SUBAPPLICATION SubApp (* Subapplication Type *)
  (* Standard: 61499-2 *)
  (* Version 1.0, 2022-12-28, kirill *)
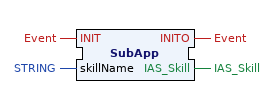
  EVENT_INPUT
    INIT;
  END_EVENT
  EVENT_OUTPUT
    INITO;
  END_EVENT
  VAR_INPUT
    skillName : STRING;
  END_VAR
  PLUGS
    IAS_Skill : IAS_Skill;
  END_PLUGS
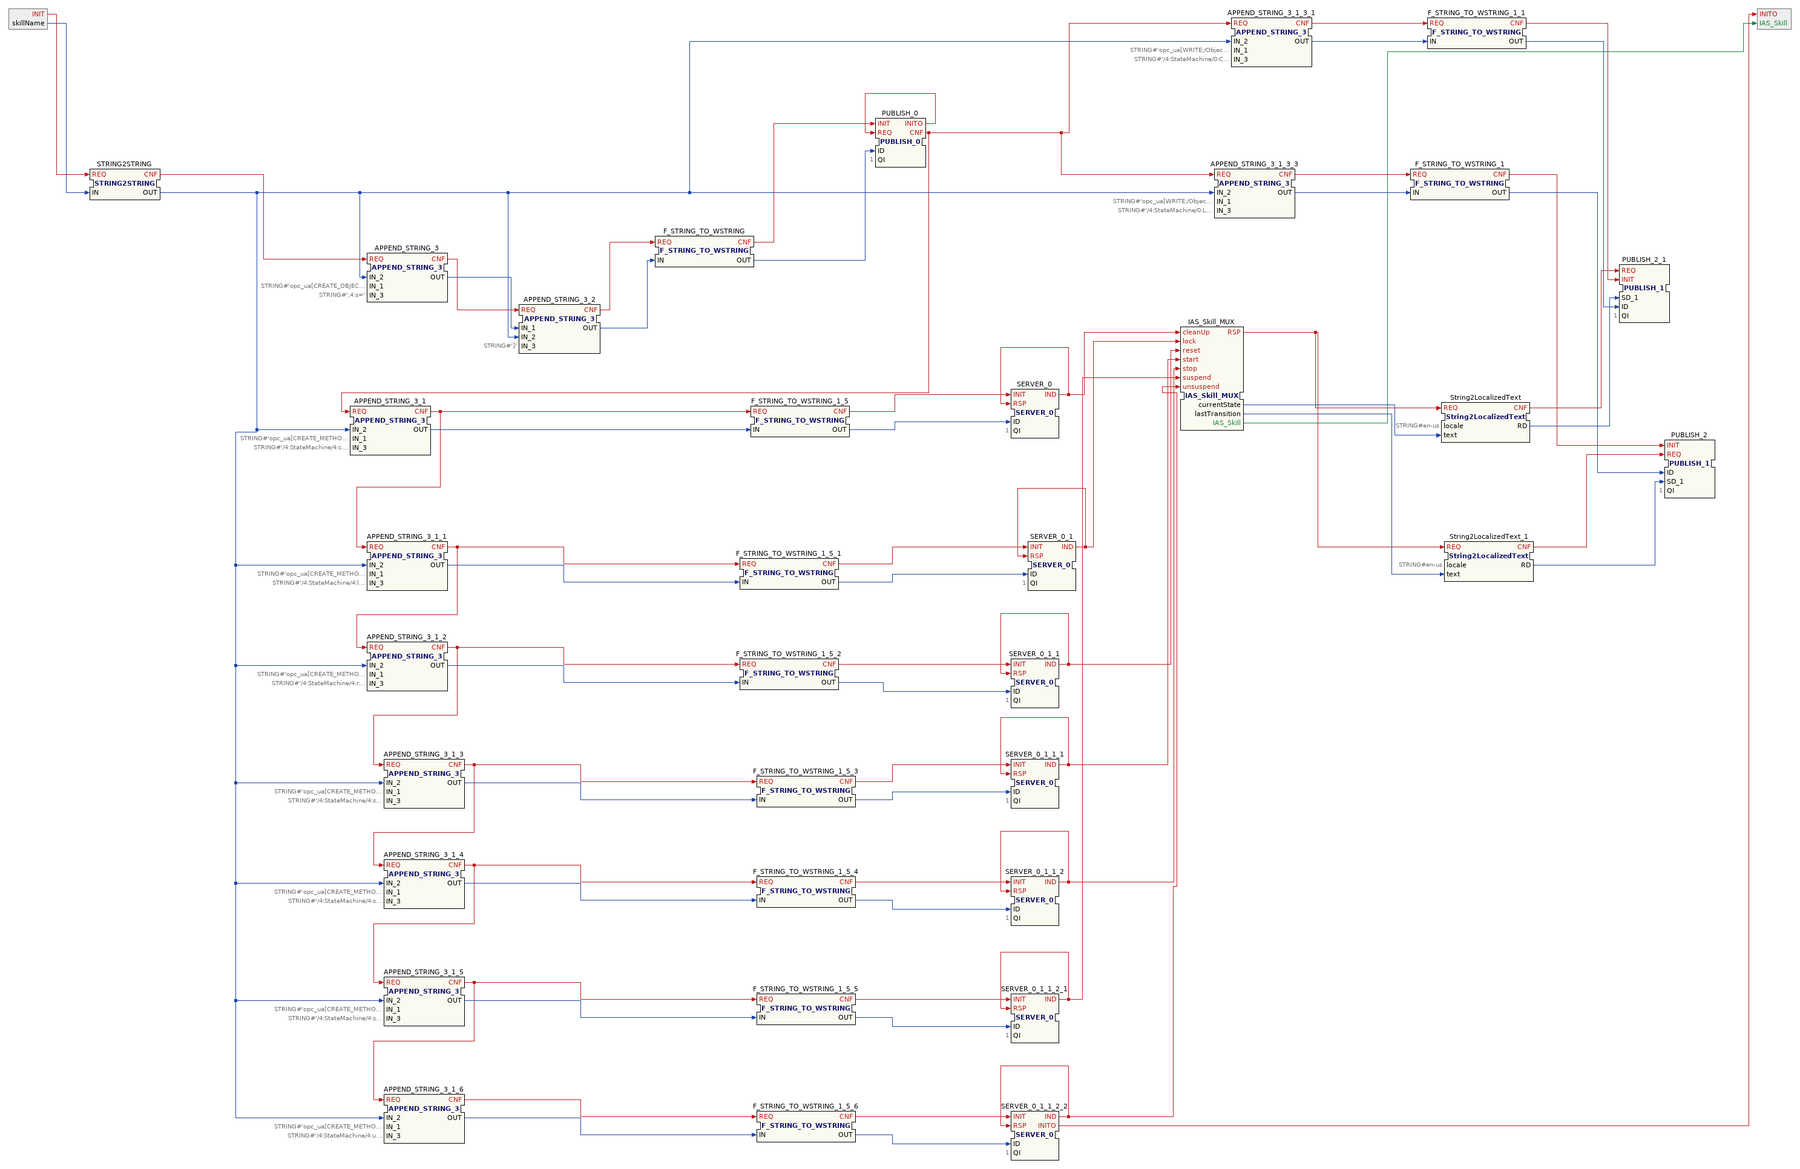
  FBS
    SERVER_0 : SERVER_0(QI := 1);
    APPEND_STRING_3 : APPEND_STRING_3(IN_1 := STRING#'opc_ua[CREATE_OBJECT;,i=58;/Objects/4:', IN_3 := STRING#',4:s=');
    PUBLISH_0 : PUBLISH_0(QI := 1);
    String2LocalizedText : String2LocalizedText(locale := STRING#en-us);
    STRING2STRING : STRING2STRING;
    SERVER_0_1_1_2 : SERVER_0(QI := 1);
    APPEND_STRING_3_1_3_1 : APPEND_STRING_3(IN_1 := STRING#'opc_ua[WRITE;/Objects/4:', IN_3 := STRING#'/4:StateMachine/0:CurrentState]');
    F_STRING_TO_WSTRING_1_5_1 : F_STRING_TO_WSTRING;
    APPEND_STRING_3_1_3_3 : APPEND_STRING_3(IN_1 := STRING#'opc_ua[WRITE;/Objects/4:', IN_3 := STRING#'/4:StateMachine/0:LastTransition]');
    F_STRING_TO_WSTRING_1_5 : F_STRING_TO_WSTRING;
    F_STRING_TO_WSTRING_1_1 : F_STRING_TO_WSTRING;
    IAS_Skill_MUX : IAS_Skill_MUX;
    APPEND_STRING_3_1_2 : APPEND_STRING_3(IN_1 := STRING#'opc_ua[CREATE_METHOD;/Objects/4:', IN_3 := STRING#'/4:StateMachine/4:reset]');
    SERVER_0_1_1_2_1 : SERVER_0(QI := 1);
    PUBLISH_2 : PUBLISH_1(QI := 1);
    SERVER_0_1_1_1 : SERVER_0(QI := 1);
    SERVER_0_1 : SERVER_0(QI := 1);
    APPEND_STRING_3_2 : APPEND_STRING_3(IN_3 := STRING#']');
    F_STRING_TO_WSTRING_1_5_5 : F_STRING_TO_WSTRING;
    SERVER_0_1_1 : SERVER_0(QI := 1);
    F_STRING_TO_WSTRING_1_5_3 : F_STRING_TO_WSTRING;
    APPEND_STRING_3_1_4 : APPEND_STRING_3(IN_1 := STRING#'opc_ua[CREATE_METHOD;/Objects/4:', IN_3 := STRING#'/4:StateMachine/4:stop]');
    APPEND_STRING_3_1_3 : APPEND_STRING_3(IN_1 := STRING#'opc_ua[CREATE_METHOD;/Objects/4:', IN_3 := STRING#'/4:StateMachine/4:start]');
    PUBLISH_2_1 : PUBLISH_1(QI := 1);
    APPEND_STRING_3_1_1 : APPEND_STRING_3(IN_1 := STRING#'opc_ua[CREATE_METHOD;/Objects/4:', IN_3 := STRING#'/4:StateMachine/4:lock]');
    F_STRING_TO_WSTRING_1_5_2 : F_STRING_TO_WSTRING;
    APPEND_STRING_3_1_6 : APPEND_STRING_3(IN_1 := STRING#'opc_ua[CREATE_METHOD;/Objects/4:', IN_3 := STRING#'/4:StateMachine/4:unsuspend]');
    F_STRING_TO_WSTRING : F_STRING_TO_WSTRING;
    SERVER_0_1_1_2_2 : SERVER_0(QI := 1);
    APPEND_STRING_3_1 : APPEND_STRING_3(IN_1 := STRING#'opc_ua[CREATE_METHOD;/Objects/4:', IN_3 := STRING#'/4:StateMachine/4:cleanUp]');
    F_STRING_TO_WSTRING_1_5_6 : F_STRING_TO_WSTRING;
    String2LocalizedText_1 : String2LocalizedText(locale := STRING#en-us);
    F_STRING_TO_WSTRING_1 : F_STRING_TO_WSTRING;
    F_STRING_TO_WSTRING_1_5_4 : F_STRING_TO_WSTRING;
    APPEND_STRING_3_1_5 : APPEND_STRING_3(IN_1 := STRING#'opc_ua[CREATE_METHOD;/Objects/4:', IN_3 := STRING#'/4:StateMachine/4:suspend]');
  END_FBS
  EVENT_CONNECTIONS
    F_STRING_TO_WSTRING_1_5.CNF TO SERVER_0.INIT;
    SERVER_0.IND TO SERVER_0.RSP;
    SERVER_0.IND TO IAS_Skill_MUX.cleanUp;
    STRING2STRING.CNF TO APPEND_STRING_3.REQ;
    APPEND_STRING_3.CNF TO APPEND_STRING_3_2.REQ;
    F_STRING_TO_WSTRING.CNF TO PUBLISH_0.INIT;
    PUBLISH_0.INITO TO PUBLISH_0.REQ;
    PUBLISH_0.CNF TO APPEND_STRING_3_1_3_3.REQ;
    PUBLISH_0.CNF TO APPEND_STRING_3_1_3_1.REQ;
    PUBLISH_0.CNF TO APPEND_STRING_3_1.REQ;
    IAS_Skill_MUX.RSP TO String2LocalizedText.REQ;
    String2LocalizedText.CNF TO PUBLISH_2_1.REQ;
    F_STRING_TO_WSTRING_1_5_4.CNF TO SERVER_0_1_1_2.INIT;
    SERVER_0_1_1_2.IND TO SERVER_0_1_1_2.RSP;
    SERVER_0_1_1_2.IND TO IAS_Skill_MUX.stop;
    APPEND_STRING_3_1_3_1.CNF TO F_STRING_TO_WSTRING_1_1.REQ;
    APPEND_STRING_3_1_1.CNF TO F_STRING_TO_WSTRING_1_5_1.REQ;
    F_STRING_TO_WSTRING_1_5_1.CNF TO SERVER_0_1.INIT;
    APPEND_STRING_3_1_3_3.CNF TO F_STRING_TO_WSTRING_1.REQ;
    APPEND_STRING_3_1.CNF TO F_STRING_TO_WSTRING_1_5.REQ;
    F_STRING_TO_WSTRING_1_1.CNF TO PUBLISH_2_1.INIT;
    SERVER_0_1.IND TO IAS_Skill_MUX.lock;
    SERVER_0_1_1.IND TO IAS_Skill_MUX.reset;
    SERVER_0_1_1_1.IND TO IAS_Skill_MUX.start;
    SERVER_0_1_1_2_1.IND TO IAS_Skill_MUX.suspend;
    SERVER_0_1_1_2_2.IND TO IAS_Skill_MUX.unsuspend;
    IAS_Skill_MUX.RSP TO String2LocalizedText_1.REQ;
    APPEND_STRING_3_1_1.CNF TO APPEND_STRING_3_1_2.REQ;
    APPEND_STRING_3_1_2.CNF TO APPEND_STRING_3_1_3.REQ;
    APPEND_STRING_3_1_2.CNF TO F_STRING_TO_WSTRING_1_5_2.REQ;
    F_STRING_TO_WSTRING_1_5_5.CNF TO SERVER_0_1_1_2_1.INIT;
    SERVER_0_1_1_2_1.IND TO SERVER_0_1_1_2_1.RSP;
    F_STRING_TO_WSTRING_1.CNF TO PUBLISH_2.INIT;
    String2LocalizedText_1.CNF TO PUBLISH_2.REQ;
    F_STRING_TO_WSTRING_1_5_3.CNF TO SERVER_0_1_1_1.INIT;
    SERVER_0_1_1_1.IND TO SERVER_0_1_1_1.RSP;
    SERVER_0_1.IND TO SERVER_0_1.RSP;
    APPEND_STRING_3_2.CNF TO F_STRING_TO_WSTRING.REQ;
    APPEND_STRING_3_1_5.CNF TO F_STRING_TO_WSTRING_1_5_5.REQ;
    F_STRING_TO_WSTRING_1_5_2.CNF TO SERVER_0_1_1.INIT;
    SERVER_0_1_1.IND TO SERVER_0_1_1.RSP;
    APPEND_STRING_3_1_3.CNF TO F_STRING_TO_WSTRING_1_5_3.REQ;
    APPEND_STRING_3_1_3.CNF TO APPEND_STRING_3_1_4.REQ;
    APPEND_STRING_3_1_4.CNF TO APPEND_STRING_3_1_5.REQ;
    APPEND_STRING_3_1_4.CNF TO F_STRING_TO_WSTRING_1_5_4.REQ;
    APPEND_STRING_3_1.CNF TO APPEND_STRING_3_1_1.REQ;
    APPEND_STRING_3_1_5.CNF TO APPEND_STRING_3_1_6.REQ;
    APPEND_STRING_3_1_6.CNF TO F_STRING_TO_WSTRING_1_5_6.REQ;
    F_STRING_TO_WSTRING_1_5_6.CNF TO SERVER_0_1_1_2_2.INIT;
    SERVER_0_1_1_2_2.IND TO SERVER_0_1_1_2_2.RSP;
    INIT TO STRING2STRING.REQ;
    SERVER_0_1_1_2_2.INITO TO INITO;
  END_CONNECTIONS
  DATA_CONNECTIONS
    F_STRING_TO_WSTRING_1_5.OUT TO SERVER_0.ID;
    STRING2STRING.OUT TO APPEND_STRING_3.IN_2;
    APPEND_STRING_3.OUT TO APPEND_STRING_3_2.IN_1;
    F_STRING_TO_WSTRING.OUT TO PUBLISH_0.ID;
    IAS_Skill_MUX.currentState TO String2LocalizedText.text;
    String2LocalizedText.RD TO PUBLISH_2_1.SD_1;
    STRING2STRING.OUT TO APPEND_STRING_3_1_3_1.IN_2;
    STRING2STRING.OUT TO APPEND_STRING_3_1.IN_2;
    STRING2STRING.OUT TO APPEND_STRING_3_1_4.IN_2;
    STRING2STRING.OUT TO APPEND_STRING_3_1_1.IN_2;
    STRING2STRING.OUT TO APPEND_STRING_3_2.IN_2;
    STRING2STRING.OUT TO APPEND_STRING_3_1_2.IN_2;
    STRING2STRING.OUT TO APPEND_STRING_3_1_6.IN_2;
    STRING2STRING.OUT TO APPEND_STRING_3_1_3.IN_2;
    STRING2STRING.OUT TO APPEND_STRING_3_1_3_3.IN_2;
    STRING2STRING.OUT TO APPEND_STRING_3_1_5.IN_2;
    F_STRING_TO_WSTRING_1_5_4.OUT TO SERVER_0_1_1_2.ID;
    APPEND_STRING_3_1_3_1.OUT TO F_STRING_TO_WSTRING_1_1.IN;
    APPEND_STRING_3_1_1.OUT TO F_STRING_TO_WSTRING_1_5_1.IN;
    F_STRING_TO_WSTRING_1_5_1.OUT TO SERVER_0_1.ID;
    APPEND_STRING_3_1_3_3.OUT TO F_STRING_TO_WSTRING_1.IN;
    APPEND_STRING_3_1.OUT TO F_STRING_TO_WSTRING_1_5.IN;
    F_STRING_TO_WSTRING_1_1.OUT TO PUBLISH_2_1.ID;
    IAS_Skill_MUX.lastTransition TO String2LocalizedText_1.text;
    APPEND_STRING_3_1_2.OUT TO F_STRING_TO_WSTRING_1_5_2.IN;
    F_STRING_TO_WSTRING_1_5_5.OUT TO SERVER_0_1_1_2_1.ID;
    F_STRING_TO_WSTRING_1.OUT TO PUBLISH_2.ID;
    String2LocalizedText_1.RD TO PUBLISH_2.SD_1;
    F_STRING_TO_WSTRING_1_5_3.OUT TO SERVER_0_1_1_1.ID;
    APPEND_STRING_3_2.OUT TO F_STRING_TO_WSTRING.IN;
    APPEND_STRING_3_1_5.OUT TO F_STRING_TO_WSTRING_1_5_5.IN;
    F_STRING_TO_WSTRING_1_5_2.OUT TO SERVER_0_1_1.ID;
    APPEND_STRING_3_1_3.OUT TO F_STRING_TO_WSTRING_1_5_3.IN;
    APPEND_STRING_3_1_4.OUT TO F_STRING_TO_WSTRING_1_5_4.IN;
    APPEND_STRING_3_1_6.OUT TO F_STRING_TO_WSTRING_1_5_6.IN;
    F_STRING_TO_WSTRING_1_5_6.OUT TO SERVER_0_1_1_2_2.ID;
    skillName TO STRING2STRING.IN;
  END_CONNECTIONS
  ADAPTER_CONNECTIONS
    IAS_Skill_MUX.IAS_Skill TO IAS_Skill;
  END_CONNECTIONS
END_SUBAPPLICATION
